(* PLC project Unnamed, Unknown Unnamed 1 *)
(* stored: creationDateTime 2026-03-06T11:23:47, modificationDateTime 2026-03-06T11:23:47 *)

PROGRAM main
  VAR
    S1 AT %IX0.0 : BOOL;
    S2 AT %IX0.1 : BOOL;
    H1 AT %QX0.0 : BOOL;
  END_VAR

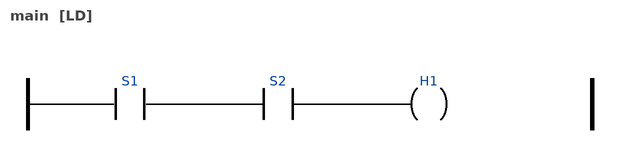
(* LD diagram, written out as Structured Text *)
H1 := S1 AND S2;
END_PROGRAM

CONFIGURATION Config0
  RESOURCE Res0 ON PLC
    TASK task0(INTERVAL := T#20ms, PRIORITY := 1);
    PROGRAM instance0 WITH task0 : main;
  END_RESOURCE
END_CONFIGURATION
